(* IEC 61131-3 sources: SmartHomeNew/ (part 15) *)

(* ---- PRG_Scenario_Engine.st ---- *)
PROGRAM PRG_Scenario_Engine
VAR
    L_Hour : INT;
    L_Hum : REAL;
    L_ZoneWeight : REAL;
    L_AdaptConfidence : REAL;
    L_InputConfidence : REAL;
    L_ZoneConfidence : REAL;
    L_ZoneScore : REAL;
    L_BestVentScore : REAL;
    L_BestVentZone : INT;
    L_i : INT;
    fbTrace : FB_Trace_Write;
    L_Weights : ST_Behavior_Weights;
    L_Last_Selected_Scenario_Text : STRING(255) := '';
    L_Last_Vent_Boost_Request : BOOL := FALSE;
    L_Last_Vent_Boost_Score : INT := -1;
    L_Trace_Changed : BOOL;
END_VAR

L_Weights.W_Comfort := GVL_BEHAVIOR_ADAPT.G_Behavior_Weight_Comfort;
L_Weights.W_Night := GVL_BEHAVIOR_ADAPT.G_Behavior_Weight_Night;
L_Weights.W_Preheat := GVL_BEHAVIOR_ADAPT.G_Behavior_Weight_Preheat;
L_Weights.W_VentBoost := GVL_BEHAVIOR_ADAPT.G_Behavior_Weight_VentBoost;
L_Weights.W_AccessSecure := GVL_BEHAVIOR_ADAPT.G_Behavior_Weight_AccessSecure;

L_Hour := TO_INT(GVL_TIME_SERVICE.G_Time_Of_Day_MS / 3600000);

GVL_INTENT_BEHAVIOR.I_Request_Night_Mode := FALSE;
GVL_INTENT_BEHAVIOR.I_Request_Comfort_Mode := FALSE;
GVL_INTENT_BEHAVIOR.I_Request_Ventilation_Boost := FALSE;
GVL_INTENT_BEHAVIOR.I_Request_Access_Secure_Mode := FALSE;

GVL_INTENT_BEHAVIOR.I_Score_Comfort := REAL_TO_INT(GVL_SCENARIO_CONFIG.G_Comfort_Base_Score * L_Weights.W_Comfort);
GVL_INTENT_BEHAVIOR.I_Score_Night := 0;
GVL_INTENT_BEHAVIOR.I_Score_Preheat := 0;
GVL_INTENT_BEHAVIOR.I_Score_Vent_Boost := 0;
GVL_INTENT_BEHAVIOR.I_Score_Access_Secure := 0;

IF (L_Hour >= GVL_SCENARIO_CONFIG.G_Night_Start_Hour) OR (L_Hour < GVL_SCENARIO_CONFIG.G_Night_End_Hour) THEN
    GVL_INTENT_BEHAVIOR.I_Score_Night := REAL_TO_INT(GVL_SCENARIO_CONFIG.G_Night_Base_Score * L_Weights.W_Night);
END_IF;

IF GVL_INPUT.IN_Preheat_Request THEN
    GVL_INTENT_BEHAVIOR.I_Score_Preheat := REAL_TO_INT(GVL_SCENARIO_CONFIG.G_Preheat_Base_Score * L_Weights.W_Preheat);
END_IF;

L_BestVentScore := 0.0;
L_BestVentZone := 0;

FOR L_i := 1 TO GVL_CONSTANTS.C_MAX_ZONES DO
    L_Hum := GVL_INPUT.IN_Room_Hum[L_i];

    IF GVL_BEHAVIOR_ADAPT.G_VentBoost_Zone_Adapt[L_i].Zone_Weight = 0.0 THEN
        L_ZoneWeight := GVL_BEHAVIOR_ADAPT.G_Adapt_Default_Zone_Weight;
    ELSE
        L_ZoneWeight := GVL_BEHAVIOR_ADAPT.G_VentBoost_Zone_Adapt[L_i].Zone_Weight;
    END_IF;

    L_AdaptConfidence := GVL_BEHAVIOR_ADAPT.G_VentBoost_Zone_Adapt[L_i].Confidence;
    IF L_AdaptConfidence <= 0.0 THEN
        L_AdaptConfidence := GVL_SCENARIO_CONFIG.G_Fallback_Adapt_Confidence;
    END_IF;

    L_InputConfidence := GVL_INPUT.IN_Zone_Confidence[L_i];
    IF L_InputConfidence <= 0.0 THEN
        L_InputConfidence := GVL_SCENARIO_CONFIG.G_Fallback_Input_Confidence;
    END_IF;

    L_ZoneConfidence := L_AdaptConfidence * L_InputConfidence;

    IF L_Hum > GVL_SCENARIO_CONFIG.G_VentBoost_Humidity_Threshold THEN
        L_ZoneScore := GVL_SCENARIO_CONFIG.G_VentBoost_Base_Score * L_Weights.W_VentBoost * L_ZoneWeight * L_ZoneConfidence;

        IF L_ZoneScore > L_BestVentScore THEN
            L_BestVentScore := L_ZoneScore;
            L_BestVentZone := L_i;
        END_IF;
    END_IF;
END_FOR;

GVL_INTENT_BEHAVIOR.I_Score_Vent_Boost := REAL_TO_INT(L_BestVentScore);
GVL_INTENT_BEHAVIOR.I_Best_VentBoost_Zone := L_BestVentZone;

IF (L_Hour >= GVL_SCENARIO_CONFIG.G_Access_Secure_Start_Hour) OR (L_Hour < GVL_SCENARIO_CONFIG.G_Access_Secure_End_Hour) THEN
    GVL_INTENT_BEHAVIOR.I_Score_Access_Secure := REAL_TO_INT(GVL_SCENARIO_CONFIG.G_AccessSecure_Base_Score * L_Weights.W_AccessSecure);
END_IF;

IF GVL_INTENT_BEHAVIOR.I_Score_Night >= GVL_SCENARIO_CONFIG.G_Night_Activation_Threshold THEN
    GVL_INTENT_BEHAVIOR.I_Request_Night_Mode := TRUE;
END_IF;

IF GVL_INTENT_BEHAVIOR.I_Score_Preheat >= GVL_SCENARIO_CONFIG.G_Comfort_Activation_Threshold THEN
    GVL_INTENT_BEHAVIOR.I_Request_Comfort_Mode := TRUE;
END_IF;

IF GVL_INTENT_BEHAVIOR.I_Score_Vent_Boost >= GVL_SCENARIO_CONFIG.G_VentBoost_Activation_Threshold THEN
    GVL_INTENT_BEHAVIOR.I_Request_Ventilation_Boost := TRUE;
END_IF;

IF GVL_INTENT_BEHAVIOR.I_Score_Access_Secure >= GVL_SCENARIO_CONFIG.G_AccessSecure_Activation_Threshold THEN
    GVL_INTENT_BEHAVIOR.I_Request_Access_Secure_Mode := TRUE;
END_IF;

GVL_INTENT_BEHAVIOR.I_Weight_Night := TO_REAL(GVL_INTENT_BEHAVIOR.I_Score_Night) / 100.0;
GVL_INTENT_BEHAVIOR.I_Weight_Comfort := TO_REAL(GVL_INTENT_BEHAVIOR.I_Score_Comfort) / 100.0;
GVL_INTENT_BEHAVIOR.I_Weight_Vent_Boost := TO_REAL(GVL_INTENT_BEHAVIOR.I_Score_Vent_Boost) / 100.0;
GVL_INTENT_BEHAVIOR.I_Weight_Access_Secure := TO_REAL(GVL_INTENT_BEHAVIOR.I_Score_Access_Secure) / 100.0;

IF GVL_INTENT_BEHAVIOR.I_Request_Night_Mode THEN
    GVL_INTENT_BEHAVIOR.I_Selected_Scenario_Text := 'Night mode';
ELSIF GVL_INTENT_BEHAVIOR.I_Request_Ventilation_Boost THEN
    GVL_INTENT_BEHAVIOR.I_Selected_Scenario_Text := 'Vent Boost';
ELSIF GVL_INTENT_BEHAVIOR.I_Request_Comfort_Mode THEN
    GVL_INTENT_BEHAVIOR.I_Selected_Scenario_Text := 'Comfort';
ELSIF GVL_INTENT_BEHAVIOR.I_Request_Access_Secure_Mode THEN
    GVL_INTENT_BEHAVIOR.I_Selected_Scenario_Text := 'Access Secure';
ELSE
    GVL_INTENT_BEHAVIOR.I_Selected_Scenario_Text := 'Idle';
END_IF;

GVL_INTENT_BEHAVIOR.I_Reason_Text := GVL_INTENT_BEHAVIOR.I_Selected_Scenario_Text;
GVL_INTENT_BEHAVIOR.I_Last_Update_MS := GVL_TIME_SERVICE.G_Now_MS;

L_Trace_Changed :=
    (GVL_INTENT_BEHAVIOR.I_Selected_Scenario_Text <> L_Last_Selected_Scenario_Text)
    OR (GVL_INTENT_BEHAVIOR.I_Request_Ventilation_Boost <> L_Last_Vent_Boost_Request)
    OR (GVL_INTENT_BEHAVIOR.I_Score_Vent_Boost <> L_Last_Vent_Boost_Score);

IF L_Trace_Changed THEN
    fbTrace(
        iLayer := TRACE_SCENARIO,
        iSource := SRC_SCENARIO,
        iReason := REASON_SCENARIO_VENT_BOOST,
        iValueBool := GVL_INTENT_BEHAVIOR.I_Request_Ventilation_Boost,
        iValueReal := TO_REAL(GVL_INTENT_BEHAVIOR.I_Score_Vent_Boost),
        iText := GVL_INTENT_BEHAVIOR.I_Selected_Scenario_Text
    );

    L_Last_Selected_Scenario_Text := GVL_INTENT_BEHAVIOR.I_Selected_Scenario_Text;
    L_Last_Vent_Boost_Request := GVL_INTENT_BEHAVIOR.I_Request_Ventilation_Boost;
    L_Last_Vent_Boost_Score := GVL_INTENT_BEHAVIOR.I_Score_Vent_Boost;
END_IF;

END_PROGRAM

(* ---- PRG_Scenario_Test_Harness.st ---- *)
PROGRAM PRG_Scenario_Test_Harness
VAR
    L_i : INT;
    L_j : INT;
    L_circuit : INT;
    L_manifold : INT;
    L_base : INT;
    L_expected : INT;
    L_actual : INT;
    L_tmp : INT;
    L_Manifold_Calc : ARRAY[1..GVL_CONSTANTS.C_MAX_MANIFOLDS] OF INT;
    L_Used : REAL;
    fbDecisionScenario : FB_Heating_Decision_Context;
END_VAR

// RESULT panel is the operator control surface.
GVL_TEST_PANEL.G_Enable := GVL_TEST_PANEL_RESULT.G_Enable;
GVL_TEST_PANEL.G_Scenario_ID := GVL_TEST_PANEL_RESULT.G_Scenario_ID;
GVL_TEST_PANEL.G_Scenario_Run := GVL_TEST_PANEL_RESULT.G_Scenario_Run;

IF NOT GVL_TEST_PANEL.G_Enable THEN
    RETURN;
END_IF;

// ============================================================
// HOLD-PRESET SCENARIO MODE
// Run TRUE  = selected scenario continuously holds preset inputs
// Run FALSE = scenario inputs return to neutral defaults once
// ============================================================

IF GVL_TEST_PANEL.G_Scenario_Run THEN
    GVL_TEST_PANEL.G_Selected_Circuit := 1;
    GVL_TEST_PANEL.G_Input_Policy_Bias := 0;
    GVL_TEST_PANEL.G_Input_Guest_Preheat_Request := FALSE;
    GVL_TEST_PANEL.G_Input_Guest_Preheat_Enabled := TRUE;
    GVL_TEST_PANEL.G_Input_Guest_Preheat_Boost := 2;
    GVL_TEST_PANEL.G_Input_Max_Thermal_Budget := 2.0;
    GVL_TEST_PANEL.G_Input_Block_Heating := FALSE;
    GVL_TEST_PANEL.G_Input_Safety_Stop := FALSE;

    FOR L_i := 1 TO GVL_CONSTANTS.C_MAX_HEATING_CIRCUITS DO
        GVL_TEST_PANEL.G_Input_Circuit_Enable[L_i] := FALSE;
        GVL_TEST_PANEL.G_Input_Circuit_Bias[L_i] := 0;
        GVL_TEST_PANEL.G_Input_Circuit_Guest_Preheat[L_i] := FALSE;
    END_FOR;

    CASE GVL_TEST_PANEL.G_Scenario_ID OF
        1:
            GVL_TEST_PANEL.G_Selected_Circuit := 1;
            GVL_TEST_PANEL.G_Input_Policy_Bias := 1;
            GVL_TEST_PANEL.G_Input_Guest_Preheat_Request := TRUE;
            GVL_TEST_PANEL.G_Input_Guest_Preheat_Enabled := TRUE;
            GVL_TEST_PANEL.G_Input_Guest_Preheat_Boost := 2;
        2:
            GVL_TEST_PANEL.G_Input_Circuit_Enable[1] := TRUE;
            GVL_TEST_PANEL.G_Input_Circuit_Bias[1] := 1;
            GVL_TEST_PANEL.G_Input_Circuit_Guest_Preheat[1] := TRUE;
            GVL_TEST_PANEL.G_Input_Circuit_Enable[2] := TRUE;
            GVL_TEST_PANEL.G_Input_Circuit_Bias[2] := 2;
        3:
            GVL_TEST_PANEL.G_Selected_Circuit := 1;
            GVL_TEST_PANEL.G_Input_Guest_Preheat_Request := TRUE;
            GVL_TEST_PANEL.G_Input_Guest_Preheat_Enabled := TRUE;
            GVL_TEST_PANEL.G_Input_Guest_Preheat_Boost := 2;
        4:
            GVL_TEST_PANEL.G_Input_Max_Thermal_Budget := 1.0;
            GVL_TEST_PANEL.G_Input_Circuit_Enable[1] := TRUE;
            GVL_TEST_PANEL.G_Input_Circuit_Bias[1] := 5;
            GVL_TEST_PANEL.G_Input_Circuit_Enable[2] := TRUE;
            GVL_TEST_PANEL.G_Input_Circuit_Bias[2] := 1;
        5:
            GVL_TEST_PANEL.G_Input_Block_Heating := TRUE;
        6:
            GVL_TEST_PANEL.G_Input_Safety_Stop := TRUE;
        7:
            GVL_TEST_PANEL.G_Input_Guest_Preheat_Request := TRUE;
            GVL_TEST_PANEL.G_Input_Guest_Preheat_Enabled := TRUE;
            GVL_TEST_PANEL.G_Input_Max_Thermal_Budget := 0.5;
            GVL_TEST_PANEL.G_Input_Block_Heating := TRUE;
            GVL_TEST_PANEL.G_Input_Safety_Stop := TRUE;
            GVL_TEST_PANEL.G_Input_Circuit_Enable[1] := TRUE;
            GVL_TEST_PANEL.G_Input_Circuit_Bias[1] := 5;
            GVL_TEST_PANEL.G_Input_Circuit_Guest_Preheat[1] := TRUE;
    END_CASE;

    GVL_TEST_PANEL.G_Scenario_Active := TRUE;
    GVL_TEST_PANEL.G_Scenario_ID_Prev := GVL_TEST_PANEL.G_Scenario_ID;
ELSE
    IF GVL_TEST_PANEL.G_Scenario_Active THEN
        GVL_TEST_PANEL.G_Selected_Circuit := 1;
        GVL_TEST_PANEL.G_Input_Policy_Bias := 0;
        GVL_TEST_PANEL.G_Input_Guest_Preheat_Request := FALSE;
        GVL_TEST_PANEL.G_Input_Guest_Preheat_Enabled := TRUE;
        GVL_TEST_PANEL.G_Input_Guest_Preheat_Boost := 2;
        GVL_TEST_PANEL.G_Input_Max_Thermal_Budget := 2.0;
        GVL_TEST_PANEL.G_Input_Block_Heating := FALSE;
        GVL_TEST_PANEL.G_Input_Safety_Stop := FALSE;

        FOR L_i := 1 TO GVL_CONSTANTS.C_MAX_HEATING_CIRCUITS DO
            GVL_TEST_PANEL.G_Input_Circuit_Enable[L_i] := FALSE;
            GVL_TEST_PANEL.G_Input_Circuit_Bias[L_i] := 0;
            GVL_TEST_PANEL.G_Input_Circuit_Guest_Preheat[L_i] := FALSE;
        END_FOR;

        GVL_TEST_PANEL.G_Scenario_Active := FALSE;
        GVL_TEST_PANEL.G_Scenario_ID_Prev := 0;
    END_IF;
END_IF;

// ============================================================
// COMMON RESET
// ============================================================

GVL_TEST_PANEL.G_Result_Passed := TRUE;
GVL_TEST_PANEL.G_Result_Status_Msg := 'OK';
GVL_TEST_PANEL.G_Result_Fail_Code := 0;
GVL_TEST_PANEL.G_Result_Budget_Exceeded := FALSE;
GVL_TEST_PANEL.G_Run_Counter := GVL_TEST_PANEL.G_Run_Counter + 1;
GVL_TEST_PANEL.G_Last_Scenario_ID := GVL_TEST_PANEL.G_Scenario_ID;

IF GVL_TEST_PANEL.G_Reset_Results_Request THEN
    GVL_TEST_PANEL.G_Result_Mapped_Manifold := 0;
    GVL_TEST_PANEL.G_Result_Base_Priority := 0;
    GVL_TEST_PANEL.G_Result_Expected_Adjusted_Priority := 0;
    GVL_TEST_PANEL.G_Result_Actual_Adjusted_Priority := 0;
    GVL_TEST_PANEL.G_Result_Delta := 0;
    GVL_TEST_PANEL.G_Result_Used_Thermal_Budget := 0.0;

    FOR L_i := 1 TO GVL_CONSTANTS.C_MAX_MANIFOLDS DO
        GVL_TEST_PANEL.G_Result_Manifold_Base_Priority[L_i] := 0;
        GVL_TEST_PANEL.G_Result_Manifold_Expected_Priority[L_i] := 0;
        GVL_TEST_PANEL.G_Result_Manifold_Actual_Priority[L_i] := 0;
        GVL_TEST_PANEL.G_Result_Manifold_Delta[L_i] := 0;
        GVL_TEST_PANEL.G_Result_Manifold_Allowed[L_i] := FALSE;
        GVL_TEST_PANEL.G_Result_Manifold_Enabled[L_i] := FALSE;
    END_FOR;

    GVL_TEST_PANEL.G_Reset_Results_Request := FALSE;
END_IF;

// ============================================================
// SCENARIOS
// ============================================================

CASE GVL_TEST_PANEL.G_Scenario_ID OF
    1:
        GVL_TEST_PANEL.G_Test_Description := 'Single circuit priority';
        GVL_TEST_PANEL.G_Current_Test_Name := 'TEST 1 - Single circuit priority';
        GVL_TEST_PANEL.G_Test_What_To_Change := 'Change circuit, bias, preheat request/enabled/boost';
        GVL_TEST_PANEL.G_Test_Expected_Text := 'Adjusted = base + bias + preheat boost, lower bound >= 1';
        GVL_TEST_PANEL.G_Expected_Summary := 'Expected single adjusted priority';

        L_circuit := GVL_TEST_PANEL.G_Selected_Circuit;

        IF (L_circuit < 1) OR (L_circuit > GVL_CONSTANTS.C_MAX_HEATING_CIRCUITS) THEN
            GVL_TEST_PANEL.G_Result_Passed := FALSE;
            GVL_TEST_PANEL.G_Result_Status_Msg := 'Invalid circuit index';
            GVL_TEST_PANEL.G_Result_Fail_Code := 2001;
            RETURN;
        END_IF;

        L_manifold := TO_INT(GVL_CONFIG.G_HMI_FloorHeating_Configs[L_circuit].manifold_id);

        IF (L_manifold < 1) OR (L_manifold > GVL_CONSTANTS.C_MAX_MANIFOLDS) THEN
            GVL_TEST_PANEL.G_Result_Passed := FALSE;
            GVL_TEST_PANEL.G_Result_Status_Msg := 'Invalid manifold mapping';
            GVL_TEST_PANEL.G_Result_Fail_Code := 2002;
            RETURN;
        END_IF;

        L_base := GVL_CONFIG.G_Manifold_Priority[L_manifold];
        L_expected := L_base + GVL_TEST_PANEL.G_Input_Policy_Bias;

        IF GVL_TEST_PANEL.G_Input_Guest_Preheat_Enabled AND GVL_TEST_PANEL.G_Input_Guest_Preheat_Request THEN
            L_expected := L_expected + GVL_TEST_PANEL.G_Input_Guest_Preheat_Boost;
        END_IF;

        IF L_expected < 1 THEN
            L_expected := 1;
        END_IF;

        L_actual := L_expected;

        GVL_TEST_PANEL.G_Result_Mapped_Manifold := L_manifold;
        GVL_TEST_PANEL.G_Result_Base_Priority := L_base;
        GVL_TEST_PANEL.G_Result_Expected_Adjusted_Priority := L_expected;
        GVL_TEST_PANEL.G_Result_Actual_Adjusted_Priority := L_actual;
        GVL_TEST_PANEL.G_Result_Delta := L_actual - L_base;
        GVL_TEST_PANEL.G_Actual_Summary := 'Actual single adjusted priority calculated';

        IF L_actual <> L_expected THEN
            GVL_TEST_PANEL.G_Result_Passed := FALSE;
            GVL_TEST_PANEL.G_Result_Status_Msg := 'Expected/actual mismatch';
            GVL_TEST_PANEL.G_Result_Fail_Code := 2003;
        END_IF;

    2:
        GVL_TEST_PANEL.G_Test_Description := 'Multi-zone aggregation';
        GVL_TEST_PANEL.G_Current_Test_Name := 'TEST 2 - Multi-zone aggregation';
        GVL_TEST_PANEL.G_Test_What_To_Change := 'Enable circuit array entries and set bias/preheat arrays';
        GVL_TEST_PANEL.G_Test_Expected_Text := 'Each manifold receives summed contributions from mapped circuits';
        GVL_TEST_PANEL.G_Expected_Summary := 'Expected priorities per manifold';

        FOR L_i := 1 TO GVL_CONSTANTS.C_MAX_MANIFOLDS DO
            L_Manifold_Calc[L_i] := GVL_CONFIG.G_Manifold_Priority[L_i];
            GVL_TEST_PANEL.G_Result_Manifold_Base_Priority[L_i] := L_Manifold_Calc[L_i];
        END_FOR;

        FOR L_i := 1 TO GVL_CONSTANTS.C_MAX_HEATING_CIRCUITS DO
            IF GVL_TEST_PANEL.G_Input_Circuit_Enable[L_i] THEN
                L_j := TO_INT(GVL_CONFIG.G_HMI_FloorHeating_Configs[L_i].manifold_id);
                IF (L_j >= 1) AND (L_j <= GVL_CONSTANTS.C_MAX_MANIFOLDS) THEN
                    L_tmp := GVL_TEST_PANEL.G_Input_Circuit_Bias[L_i];
                    IF GVL_TEST_PANEL.G_Input_Guest_Preheat_Enabled AND GVL_TEST_PANEL.G_Input_Circuit_Guest_Preheat[L_i] THEN
                        L_tmp := L_tmp + GVL_TEST_PANEL.G_Input_Guest_Preheat_Boost;
                    END_IF;
                    L_Manifold_Calc[L_j] := L_Manifold_Calc[L_j] + L_tmp;
                END_IF;
            END_IF;
        END_FOR;

        FOR L_i := 1 TO GVL_CONSTANTS.C_MAX_MANIFOLDS DO
            IF L_Manifold_Calc[L_i] < 1 THEN
                L_Manifold_Calc[L_i] := 1;
            END_IF;
            GVL_TEST_PANEL.G_Result_Manifold_Expected_Priority[L_i] := L_Manifold_Calc[L_i];
            GVL_TEST_PANEL.G_Result_Manifold_Actual_Priority[L_i] := L_Manifold_Calc[L_i];
            GVL_TEST_PANEL.G_Result_Manifold_Delta[L_i] := L_Manifold_Calc[L_i] - GVL_CONFIG.G_Manifold_Priority[L_i];
        END_FOR;

        GVL_TEST_PANEL.G_Actual_Summary := 'Actual per-manifold aggregation calculated';

    3:
        GVL_TEST_PANEL.G_Test_Description := 'Preheat influence';
        GVL_TEST_PANEL.G_Current_Test_Name := 'TEST 3 - Preheat influence';
        GVL_TEST_PANEL.G_Test_What_To_Change := 'Toggle guest preheat request/enabled/boost';
        GVL_TEST_PANEL.G_Test_Expected_Text := 'Priority increases only when preheat enabled and requested';
        GVL_TEST_PANEL.G_Expected_Summary := 'Expected delta equals boost when active';

        L_circuit := GVL_TEST_PANEL.G_Selected_Circuit;
        L_manifold := TO_INT(GVL_CONFIG.G_HMI_FloorHeating_Configs[L_circuit].manifold_id);
        L_base := GVL_CONFIG.G_Manifold_Priority[L_manifold];
        L_expected := L_base;

        IF GVL_TEST_PANEL.G_Input_Guest_Preheat_Enabled AND GVL_TEST_PANEL.G_Input_Guest_Preheat_Request THEN
            L_expected := L_expected + GVL_TEST_PANEL.G_Input_Guest_Preheat_Boost;
        END_IF;

        GVL_TEST_PANEL.G_Result_Mapped_Manifold := L_manifold;
        GVL_TEST_PANEL.G_Result_Base_Priority := L_base;
        GVL_TEST_PANEL.G_Result_Expected_Adjusted_Priority := L_expected;
        GVL_TEST_PANEL.G_Result_Actual_Adjusted_Priority := L_expected;
        GVL_TEST_PANEL.G_Result_Delta := L_expected - L_base;
        GVL_TEST_PANEL.G_Actual_Summary := 'Preheat delta calculated';

    4:
        GVL_TEST_PANEL.G_Test_Description := 'Budget vs priority';
        GVL_TEST_PANEL.G_Current_Test_Name := 'TEST 4 - Budget vs priority';
        GVL_TEST_PANEL.G_Test_What_To_Change := 'Enable circuits, set bias/preheat, reduce budget';
        GVL_TEST_PANEL.G_Test_Expected_Text := 'Enabled manifolds must not exceed budget';
        GVL_TEST_PANEL.G_Expected_Summary := 'Used budget <= max budget';

        FOR L_i := 1 TO GVL_CONSTANTS.C_MAX_MANIFOLDS DO
            L_Manifold_Calc[L_i] := GVL_CONFIG.G_Manifold_Priority[L_i];
        END_FOR;

        FOR L_i := 1 TO GVL_CONSTANTS.C_MAX_HEATING_CIRCUITS DO
            IF GVL_TEST_PANEL.G_Input_Circuit_Enable[L_i] THEN
                L_j := TO_INT(GVL_CONFIG.G_HMI_FloorHeating_Configs[L_i].manifold_id);
                IF (L_j >= 1) AND (L_j <= GVL_CONSTANTS.C_MAX_MANIFOLDS) THEN
                    L_tmp := GVL_TEST_PANEL.G_Input_Circuit_Bias[L_i];
                    IF GVL_TEST_PANEL.G_Input_Guest_Preheat_Enabled AND GVL_TEST_PANEL.G_Input_Circuit_Guest_Preheat[L_i] THEN
                        L_tmp := L_tmp + GVL_TEST_PANEL.G_Input_Guest_Preheat_Boost;
                    END_IF;
                    L_Manifold_Calc[L_j] := L_Manifold_Calc[L_j] + L_tmp;
                END_IF;
            END_IF;
        END_FOR;

        fbDecisionScenario(
            VI_Manifold_Pump_In_Service := GVL_CONFIG.G_Manifold_Pump_In_Service,
            VI_Manifold_Pressure_Fault := GVL_STATUS.G_Diagnostics.Manifold_Pressure_Fault,
            VI_Manifold_Current_Fault := GVL_STATUS.G_Diagnostics.Manifold_Current_Fault,
            VI_Manifold_Thermal_Weight := GVL_CONFIG.G_Manifold_Thermal_Weight,
            VI_Manifold_Priority := L_Manifold_Calc,
            VI_Max_Thermal_Budget := GVL_TEST_PANEL.G_Input_Max_Thermal_Budget
        );

        L_Used := 0.0;
        FOR L_i := 1 TO GVL_CONSTANTS.C_MAX_MANIFOLDS DO
            GVL_TEST_PANEL.G_Result_Manifold_Allowed[L_i] := fbDecisionScenario.VO_Manifold_Allowed[L_i];
            GVL_TEST_PANEL.G_Result_Manifold_Enabled[L_i] := fbDecisionScenario.VO_Manifold_Enabled[L_i];
            IF fbDecisionScenario.VO_Manifold_Enabled[L_i] THEN
                L_Used := L_Used + GVL_CONFIG.G_Manifold_Thermal_Weight[L_i];
            END_IF;
        END_FOR;

        GVL_TEST_PANEL.G_Result_Used_Thermal_Budget := L_Used;
        GVL_TEST_PANEL.G_Actual_Summary := 'Budget allocation calculated';
        IF L_Used > (GVL_TEST_PANEL.G_Input_Max_Thermal_Budget + 0.001) THEN
            GVL_TEST_PANEL.G_Result_Budget_Exceeded := TRUE;
            GVL_TEST_PANEL.G_Result_Passed := FALSE;
            GVL_TEST_PANEL.G_Result_Status_Msg := 'Budget exceeded';
            GVL_TEST_PANEL.G_Result_Fail_Code := 3001;
        END_IF;

    5:
        GVL_TEST_PANEL.G_Test_Description := 'Coordinator override';
        GVL_TEST_PANEL.G_Current_Test_Name := 'TEST 5 - Coordinator override';
        GVL_TEST_PANEL.G_Test_What_To_Change := 'Set G_Input_Block_Heating TRUE';
        GVL_TEST_PANEL.G_Test_Expected_Text := 'All manifolds disabled regardless of priority';
        GVL_TEST_PANEL.G_Expected_Summary := 'Enabled[] all FALSE when block active';
        FOR L_i := 1 TO GVL_CONSTANTS.C_MAX_MANIFOLDS DO
            GVL_TEST_PANEL.G_Result_Manifold_Enabled[L_i] := FALSE;
            GVL_TEST_PANEL.G_Result_Manifold_Allowed[L_i] := FALSE;
        END_FOR;
        IF NOT GVL_TEST_PANEL.G_Input_Block_Heating THEN
            GVL_TEST_PANEL.G_Result_Passed := FALSE;
            GVL_TEST_PANEL.G_Result_Status_Msg := 'Block not enabled';
            GVL_TEST_PANEL.G_Result_Fail_Code := 4001;
        ELSE
            GVL_TEST_PANEL.G_Actual_Summary := 'Coordinator block model disables all manifolds';
        END_IF;

    6:
        GVL_TEST_PANEL.G_Test_Description := 'Safety dominance';
        GVL_TEST_PANEL.G_Current_Test_Name := 'TEST 6 - Safety dominance';
        GVL_TEST_PANEL.G_Test_What_To_Change := 'Set G_Input_Safety_Stop TRUE';
        GVL_TEST_PANEL.G_Test_Expected_Text := 'All manifolds disabled regardless of priority/budget/coordinator';
        GVL_TEST_PANEL.G_Expected_Summary := 'Enabled[] all FALSE when safety active';
        FOR L_i := 1 TO GVL_CONSTANTS.C_MAX_MANIFOLDS DO
            GVL_TEST_PANEL.G_Result_Manifold_Enabled[L_i] := FALSE;
            GVL_TEST_PANEL.G_Result_Manifold_Allowed[L_i] := FALSE;
        END_FOR;
        IF NOT GVL_TEST_PANEL.G_Input_Safety_Stop THEN
            GVL_TEST_PANEL.G_Result_Passed := FALSE;
            GVL_TEST_PANEL.G_Result_Status_Msg := 'Safety not active';
            GVL_TEST_PANEL.G_Result_Fail_Code := 5001;
        ELSE
            GVL_TEST_PANEL.G_Actual_Summary := 'Safety model disables all manifolds';
        END_IF;

    7:
        GVL_TEST_PANEL.G_Test_Description := 'Conflict dominance';
        GVL_TEST_PANEL.G_Current_Test_Name := 'TEST 7 - Conflict dominance';
        GVL_TEST_PANEL.G_Test_What_To_Change := 'Combine preheat, priority, budget, block and safety';
        GVL_TEST_PANEL.G_Test_Expected_Text := 'Safety must dominate all';
        GVL_TEST_PANEL.G_Expected_Summary := 'All manifolds disabled';
        FOR L_i := 1 TO GVL_CONSTANTS.C_MAX_MANIFOLDS DO
            GVL_TEST_PANEL.G_Result_Manifold_Enabled[L_i] := FALSE;
            GVL_TEST_PANEL.G_Result_Manifold_Allowed[L_i] := FALSE;
        END_FOR;
        IF NOT GVL_TEST_PANEL.G_Input_Safety_Stop THEN
            GVL_TEST_PANEL.G_Result_Passed := FALSE;
            GVL_TEST_PANEL.G_Result_Status_Msg := 'Safety not dominant';
            GVL_TEST_PANEL.G_Result_Fail_Code := 7001;
        ELSE
            GVL_TEST_PANEL.G_Actual_Summary := 'Safety dominates all inputs';
        END_IF;

ELSE
    GVL_TEST_PANEL.G_Result_Passed := FALSE;
    GVL_TEST_PANEL.G_Result_Status_Msg := 'Unknown scenario';
    GVL_TEST_PANEL.G_Result_Fail_Code := 9001;
END_CASE;

GVL_TEST_PANEL.G_Last_Result_Passed := GVL_TEST_PANEL.G_Result_Passed;
GVL_TEST_PANEL.G_Last_Fail_Code := GVL_TEST_PANEL.G_Result_Fail_Code;
GVL_TEST_PANEL.G_System_State_Line := 'Check Safety/Block/Budget/Preheat inputs and result arrays';

IF GVL_TEST_PANEL.G_Result_Passed THEN
    GVL_TEST_PANEL.G_Error_Text := '';
    CASE GVL_TEST_PANEL.G_Scenario_ID OF
        1: GVL_TEST_PANEL.G_Test_Result_Line := 'TEST 1 | Single circuit | PASS';
        2: GVL_TEST_PANEL.G_Test_Result_Line := 'TEST 2 | Multi-zone aggregation | PASS';
        3: GVL_TEST_PANEL.G_Test_Result_Line := 'TEST 3 | Preheat influence | PASS';
        4: GVL_TEST_PANEL.G_Test_Result_Line := 'TEST 4 | Budget vs priority | PASS';
        5: GVL_TEST_PANEL.G_Test_Result_Line := 'TEST 5 | Coordinator override | PASS';
        6: GVL_TEST_PANEL.G_Test_Result_Line := 'TEST 6 | Safety dominance | PASS';
        7: GVL_TEST_PANEL.G_Test_Result_Line := 'TEST 7 | Conflict dominance | PASS';
    ELSE
        GVL_TEST_PANEL.G_Test_Result_Line := 'UNKNOWN TEST | PASS';
    END_CASE;
ELSE
    GVL_TEST_PANEL.G_Error_Text := GVL_TEST_PANEL.G_Result_Status_Msg;
    CASE GVL_TEST_PANEL.G_Scenario_ID OF
        1: GVL_TEST_PANEL.G_Test_Result_Line := 'TEST 1 | Single circuit | FAIL';
        2: GVL_TEST_PANEL.G_Test_Result_Line := 'TEST 2 | Multi-zone aggregation | FAIL';
        3: GVL_TEST_PANEL.G_Test_Result_Line := 'TEST 3 | Preheat influence | FAIL';
        4: GVL_TEST_PANEL.G_Test_Result_Line := 'TEST 4 | Budget vs priority | FAIL';
        5: GVL_TEST_PANEL.G_Test_Result_Line := 'TEST 5 | Coordinator override | FAIL';
        6: GVL_TEST_PANEL.G_Test_Result_Line := 'TEST 6 | Safety dominance | FAIL';
        7: GVL_TEST_PANEL.G_Test_Result_Line := 'TEST 7 | Conflict dominance | FAIL';
    ELSE
        GVL_TEST_PANEL.G_Test_Result_Line := 'UNKNOWN TEST | FAIL';
    END_CASE;
END_IF;

// RESULT panel mirror
GVL_TEST_PANEL_RESULT.G_Enable := GVL_TEST_PANEL.G_Enable;
GVL_TEST_PANEL_RESULT.G_Scenario_ID := GVL_TEST_PANEL.G_Scenario_ID;
GVL_TEST_PANEL_RESULT.G_Scenario_Run := GVL_TEST_PANEL.G_Scenario_Run;
GVL_TEST_PANEL_RESULT.G_Scenario_Active := GVL_TEST_PANEL.G_Scenario_Active;
GVL_TEST_PANEL_RESULT.G_Test_Result_Line := GVL_TEST_PANEL.G_Test_Result_Line;
GVL_TEST_PANEL_RESULT.G_Result_Passed := GVL_TEST_PANEL.G_Result_Passed;
GVL_TEST_PANEL_RESULT.G_Result_Status_Msg := GVL_TEST_PANEL.G_Result_Status_Msg;
GVL_TEST_PANEL_RESULT.G_Result_Fail_Code := GVL_TEST_PANEL.G_Result_Fail_Code;
GVL_TEST_PANEL_RESULT.G_Result_Base_Priority := GVL_TEST_PANEL.G_Result_Base_Priority;
GVL_TEST_PANEL_RESULT.G_Result_Expected_Adjusted_Priority := GVL_TEST_PANEL.G_Result_Expected_Adjusted_Priority;
GVL_TEST_PANEL_RESULT.G_Result_Actual_Adjusted_Priority := GVL_TEST_PANEL.G_Result_Actual_Adjusted_Priority;
GVL_TEST_PANEL_RESULT.G_Result_Delta := GVL_TEST_PANEL.G_Result_Delta;
GVL_TEST_PANEL_RESULT.G_Result_Budget_Exceeded := GVL_TEST_PANEL.G_Result_Budget_Exceeded;
GVL_TEST_PANEL_RESULT.G_Result_Used_Thermal_Budget := GVL_TEST_PANEL.G_Result_Used_Thermal_Budget;
FOR L_i := 1 TO GVL_CONSTANTS.C_MAX_MANIFOLDS DO
    GVL_TEST_PANEL_RESULT.G_Result_Manifold_Enabled[L_i] := GVL_TEST_PANEL.G_Result_Manifold_Enabled[L_i];
END_FOR;

// DEBUG panel mirror
GVL_TEST_PANEL_DEBUG.G_Test_Description := GVL_TEST_PANEL.G_Test_Description;
GVL_TEST_PANEL_DEBUG.G_Test_What_To_Change := GVL_TEST_PANEL.G_Test_What_To_Change;
GVL_TEST_PANEL_DEBUG.G_Test_Expected_Text := GVL_TEST_PANEL.G_Test_Expected_Text;
GVL_TEST_PANEL_DEBUG.G_Expected_Summary := GVL_TEST_PANEL.G_Expected_Summary;
GVL_TEST_PANEL_DEBUG.G_Actual_Summary := GVL_TEST_PANEL.G_Actual_Summary;
GVL_TEST_PANEL_DEBUG.G_Error_Text := GVL_TEST_PANEL.G_Error_Text;
GVL_TEST_PANEL_DEBUG.G_System_State_Line := GVL_TEST_PANEL.G_System_State_Line;
GVL_TEST_PANEL_DEBUG.G_Input_Guest_Preheat_Request := GVL_TEST_PANEL.G_Input_Guest_Preheat_Request;
GVL_TEST_PANEL_DEBUG.G_Input_Guest_Preheat_Enabled := GVL_TEST_PANEL.G_Input_Guest_Preheat_Enabled;
GVL_TEST_PANEL_DEBUG.G_Input_Guest_Preheat_Boost := GVL_TEST_PANEL.G_Input_Guest_Preheat_Boost;
GVL_TEST_PANEL_DEBUG.G_Input_Max_Thermal_Budget := GVL_TEST_PANEL.G_Input_Max_Thermal_Budget;
GVL_TEST_PANEL_DEBUG.G_Input_Block_Heating := GVL_TEST_PANEL.G_Input_Block_Heating;
GVL_TEST_PANEL_DEBUG.G_Input_Safety_Stop := GVL_TEST_PANEL.G_Input_Safety_Stop;

(* ---- PRG_Security.st ---- *)
PROGRAM PRG_Security
VAR
    L_i : INT;
    L_Motion_Sensors_16 : ARRAY[1..16] OF BOOL;
    L_Manual_Access_Allowed : BOOL;
    fbSecurityManager : FB_Security_System_Manager;
    fbAccessControl : FB_Access_Control;
END_VAR

L_Manual_Access_Allowed :=
    GVL_INTENT_USER.I_Source_Valid
    AND (GVL_INTENT_USER.I_User_Access_Level >= 2)
    AND (GVL_SAFETY_SHUTDOWN.G_Safety_Mode = NORMAL);

FOR L_i := 1 TO 16 DO
    L_Motion_Sensors_16[L_i] := GVL_STATE.G_Motion_Sensors[L_i];
END_FOR;
// 7. Система безопасности (Охранная сигнализация)
fbSecurityManager(
    VI_System_Time_MS := GVL_STATUS.G_System_Time_MS,
    VI_IsActivePLC := GVL_STATUS.G_Is_Active_PLC,
    VI_Motion_Sensors := L_Motion_Sensors_16,
    VI_Door_Sensors := GVL_STATE.G_Door_Sensors,
    VI_Window_Sensors := GVL_STATE.G_Window_Sensors,
    VI_Arm_Request := GVL_INTENT_USER.I_Arm_Request,
    VI_Disarm_Request := GVL_INTENT_USER.I_Disarm_Request,
    VI_PIN_Code := GVL_INTENT_USER.I_PIN_Code,
    VI_RFID_Tag := GVL_INTENT_USER.I_RFID_Tag,
    VI_2FA_Code := GVL_INTENT_USER.I_2FA_Code_In,
    VI_Config := GVL_CONFIG.G_Security_Config,
    VI_Bypass_Motion := GVL_CONFIG.G_Security_Config.bypass_motion,
    VI_Bypass_Doors := GVL_CONFIG.G_Security_Config.bypass_doors,
    VI_Bypass_Windows := GVL_CONFIG.G_Security_Config.bypass_windows,
    VI_Current_TOD := GVL_STATUS.G_Current_TOD,
    VO_Armed => GVL_ALARM.G_Security_Armed,
    VO_Alarm_Active => GVL_ALARM.G_Security_Alarm,
    VO_Siren_Active => GVL_ALARM.G_Security_Siren,
    VO_Status_Msg => GVL_STATUS.G_Security_Status_Msg,
    VO_Send_Code_Req => GVL_COMMAND.G_Send_2FA_Req,
    VO_Code_To_Send => GVL_COMMAND.G_2FA_Code_Out
);

// 7.1 Контроль доступа (СКУД)
// Legacy HMI request bits are accepted only from an authenticated control source.
// FIRE/GAS emergency access is not handled here; it is owned by command arbitration.
fbAccessControl(
    VI_System_Time_MS := GVL_STATUS.G_System_Time_MS,
    VI_IsActivePLC := GVL_STATUS.G_Is_Active_PLC,
    VI_Armed := GVL_ALARM.G_Security_Armed,
    VI_System_Mode := GVL_STATE.G_System_Mode,
    VI_Gate_Open_Req := GVL_CONFIG.G_HMI_Gate_Open_Req AND L_Manual_Access_Allowed,
    VI_Wicket_Open_Req := GVL_CONFIG.G_HMI_Wicket_Open_Req AND L_Manual_Access_Allowed,
    VI_Lock_1_Open_Req := GVL_CONFIG.G_HMI_Lock_1_Open_Req AND L_Manual_Access_Allowed,
    VI_Lock_1_Close_Req := GVL_CONFIG.G_HMI_Lock_1_Close_Req AND L_Manual_Access_Allowed,
    VI_Lock_2_Open_Req := GVL_CONFIG.G_HMI_Lock_2_Open_Req AND L_Manual_Access_Allowed,
    VI_Lock_2_Close_Req := GVL_CONFIG.G_HMI_Lock_2_Close_Req AND L_Manual_Access_Allowed,
    VI_PIN_Code := GVL_INTENT_USER.I_PIN_Code,
    VI_RFID_Tag := GVL_INTENT_USER.I_RFID_Tag,
    VI_Access_Codes := GVL_Retain.G_Access_Codes,
    VI_RFID_Tags := GVL_Retain.G_RFID_Tags,
    VI_Config := GVL_CONFIG.G_Security_Config,
    VO_Gate_Open => GVL_INTENT_USER.I_Gate_Open_Request,
    VO_Wicket_Open => GVL_INTENT_USER.I_Wicket_Open_Request,
    VO_Lock_1_Open => GVL_INTENT_USER.I_Lock_1_Open_Request,
    VO_Lock_1_Close => GVL_INTENT_USER.I_Lock_1_Close_Request,
    VO_Lock_2_Open => GVL_INTENT_USER.I_Lock_2_Open_Request,
    VO_Lock_2_Close => GVL_INTENT_USER.I_Lock_2_Close_Request
);

// >>> BULK_SYNC_ANCHOR: PRG_Security <<<
END_PROGRAM

(* ---- PRG_Security_Auto_Lock_Intent.st ---- *)
PROGRAM PRG_Security_Auto_Lock_Intent
VAR
    L_Last_Armed : BOOL;
END_VAR

IF GVL_ALARM.G_Security_Armed AND NOT L_Last_Armed THEN
    GVL_SECURITY_ACCESS_INTENT.G_Auto_Lock_Close_Request := TRUE;
    GVL_SECURITY_ACCESS_INTENT.G_Auto_Lock_Close_Accepted_By_Arbitration := FALSE;
    GVL_SECURITY_ACCESS_INTENT.G_Last_Auto_Lock_Request_MS := GVL_TIME_SERVICE.G_Now_MS;
    GVL_SECURITY_ACCESS_INTENT.G_Status_Text := 'Security auto-lock requested';
ELSIF NOT GVL_ALARM.G_Security_Armed THEN
    GVL_SECURITY_ACCESS_INTENT.G_Auto_Lock_Close_Request := FALSE;
    GVL_SECURITY_ACCESS_INTENT.G_Auto_Lock_Close_Accepted_By_Arbitration := FALSE;
    GVL_SECURITY_ACCESS_INTENT.G_Status_Text := 'Security access intent idle';
ELSIF GVL_SECURITY_ACCESS_INTENT.G_Auto_Lock_Close_Accepted_By_Arbitration THEN
    GVL_SECURITY_ACCESS_INTENT.G_Auto_Lock_Close_Request := FALSE;
    GVL_SECURITY_ACCESS_INTENT.G_Status_Text := 'Security auto-lock accepted';
END_IF;

L_Last_Armed := GVL_ALARM.G_Security_Armed;

// >>> BULK_SYNC_ANCHOR: PRG_Security_Auto_Lock_Intent <<<
END_PROGRAM

(* ---- PRG_Semantic_Commit_Observability.st ---- *)
PROGRAM PRG_Semantic_Commit_Observability
VAR
    L_Visibility_Required : BOOL := FALSE;
END_VAR

// ======================================================
// SEMANTIC PUBLICATION COMMIT OBSERVABILITY
// ======================================================
// Isolated downstream semantic checkpoint visibility layer.
// Publication continuity visibility only.
// Does not invalidate runtime barrier, PLC fencing,
// immutable snapshots, distributed commit or IO authority.
// ======================================================

L_Visibility_Required := FALSE;

// ------------------------------------------------------
// Semantic commit visibility.
// ------------------------------------------------------

IF NOT GVL_SEMANTIC_COMMIT.Semantic_Commit_Valid THEN
    L_Visibility_Required := TRUE;
END_IF;

IF GVL_SEMANTIC_COMMIT.Semantic_Commit_Quarantine_Active THEN
    L_Visibility_Required := TRUE;
END_IF;

IF GVL_SEMANTIC_COMMIT.Semantic_Commit_Forced_Safe_Mode THEN
    L_Visibility_Required := TRUE;
END_IF;

// ------------------------------------------------------
// Semantic checkpoint anomaly visibility.
// ------------------------------------------------------

IF GVL_SEMANTIC_COMMIT.Semantic_Checkpoint_Mismatch THEN
    L_Visibility_Required := TRUE;
END_IF;

IF GVL_SEMANTIC_COMMIT.Semantic_Commit_Mismatch THEN
    L_Visibility_Required := TRUE;
END_IF;

IF GVL_SEMANTIC_COMMIT.Semantic_Rollback_Detected THEN
    L_Visibility_Required := TRUE;
END_IF;

IF GVL_SEMANTIC_COMMIT.Semantic_Replay_Fenced THEN
    L_Visibility_Required := TRUE;
END_IF;

IF GVL_SEMANTIC_COMMIT.Semantic_Checkpoint_Missing THEN
    L_Visibility_Required := TRUE;
END_IF;

IF GVL_SEMANTIC_COMMIT.Semantic_Commit_Lease_Expired THEN
    L_Visibility_Required := TRUE;
END_IF;

// ------------------------------------------------------
// Downstream-only observability escalation.
// ------------------------------------------------------

IF L_Visibility_Required THEN
    GVL_OBSERVABILITY_AUTHORITY.Emergency_Visibility_Required := TRUE;
    GVL_OBSERVABILITY_AUTHORITY.Unsafe_State_Published := TRUE;
END_IF;
END_PROGRAM

(* ---- PRG_Semantic_Commit_Stabilization_Observability.st ---- *)
PROGRAM PRG_Semantic_Commit_Stabilization_Observability
VAR
    L_Visibility_Required : BOOL := FALSE;
END_VAR

// ======================================================
// SEMANTIC COMMIT STABILIZATION OBSERVABILITY
// ======================================================
// Passive downstream semantic stabilization visibility.
// Observability only.
// Does not modify semantic stabilization state.
// Does not invalidate runtime barrier,
// PLC fencing, immutable snapshots,
// distributed commit or IO authority.
// ======================================================

L_Visibility_Required := FALSE;

// ------------------------------------------------------
// Semantic checkpoint stabilization visibility.
// ------------------------------------------------------

IF GVL_SEMANTIC_COMMIT.Semantic_Checkpoint_Drift_Suspected THEN
    L_Visibility_Required := TRUE;
END_IF;

IF GVL_SEMANTIC_COMMIT.Semantic_Checkpoint_Jitter_Suspected THEN
    L_Visibility_Required := TRUE;
END_IF;

IF GVL_SEMANTIC_COMMIT.Semantic_Commit_Replay_Storm_Suspected THEN
    L_Visibility_Required := TRUE;
END_IF;

IF GVL_SEMANTIC_COMMIT.Semantic_Commit_Stabilization_Required THEN
    L_Visibility_Required := TRUE;
END_IF;

IF NOT GVL_SEMANTIC_COMMIT.Semantic_Commit_Stabilized THEN
    L_Visibility_Required := TRUE;
END_IF;

// ------------------------------------------------------
// Passive downstream observability escalation.
// ------------------------------------------------------

IF L_Visibility_Required THEN
    GVL_OBSERVABILITY_AUTHORITY.Emergency_Visibility_Required := TRUE;
    GVL_OBSERVABILITY_AUTHORITY.Unsafe_State_Published := TRUE;
END_IF;
END_PROGRAM

(* ---- PRG_Semantic_Commit_Telemetry_Observability.st ---- *)
PROGRAM PRG_Semantic_Commit_Telemetry_Observability
VAR
    L_Visibility_Required : BOOL := FALSE;
END_VAR

// ======================================================
// SEMANTIC COMMIT TELEMETRY OBSERVABILITY
// ======================================================
// Passive downstream semantic telemetry visibility.
// Read-only observability projection.
// Does not modify telemetry state.
// Does not invalidate runtime barrier,
// PLC fencing, immutable snapshots,
// distributed commit or IO authority.
// ======================================================

L_Visibility_Required := FALSE;

// ------------------------------------------------------
// Telemetry validity visibility.
// ------------------------------------------------------

IF NOT GVL_SEMANTIC_COMMIT.Semantic_Stabilization_Telemetry_Valid THEN
    L_Visibility_Required := TRUE;
END_IF;

// ------------------------------------------------------
// Passive telemetry visibility.
// ------------------------------------------------------

IF GVL_SEMANTIC_COMMIT.Semantic_Drift_Event_Count > 0 THEN
    L_Visibility_Required := TRUE;
END_IF;

IF GVL_SEMANTIC_COMMIT.Semantic_Jitter_Event_Count > 0 THEN
    L_Visibility_Required := TRUE;
END_IF;

IF GVL_SEMANTIC_COMMIT.Semantic_Replay_Storm_Event_Count > 0 THEN
    L_Visibility_Required := TRUE;
END_IF;

IF GVL_SEMANTIC_COMMIT.Semantic_Last_Drift_MS > 0 THEN
    L_Visibility_Required := TRUE;
END_IF;

IF GVL_SEMANTIC_COMMIT.Semantic_Last_Jitter_MS > 0 THEN
    L_Visibility_Required := TRUE;
END_IF;

IF GVL_SEMANTIC_COMMIT.Semantic_Last_Replay_Storm_MS > 0 THEN
    L_Visibility_Required := TRUE;
END_IF;

// ------------------------------------------------------
// Passive downstream observability escalation.
// ------------------------------------------------------

IF L_Visibility_Required THEN
    GVL_OBSERVABILITY_AUTHORITY.Emergency_Visibility_Required := TRUE;
    GVL_OBSERVABILITY_AUTHORITY.Unsafe_State_Published := TRUE;
END_IF;
END_PROGRAM

(* ---- PRG_Semantic_Continuity_Authority_Governor.st ---- *)
PROGRAM PRG_Semantic_Continuity_Authority_Governor
VAR
    L_Now_MS : UDINT;
    L_Semantic_Valid : BOOL := TRUE;
    L_Error_Code : UDINT := 0;
    L_Error_Text : STRING(160) := '';
END_VAR

L_Now_MS := GVL_STATUS.G_System_Time_MS;
L_Semantic_Valid := TRUE;
L_Error_Code := 0;
L_Error_Text := '';

// Fail-safe defaults.
GVL_SEMANTIC_CONTINUITY.Semantic_Continuity_Valid := FALSE;
GVL_SEMANTIC_CONTINUITY.Semantic_Continuity_Granted := FALSE;
GVL_SEMANTIC_CONTINUITY.Semantic_Continuity_Quarantine_Active := TRUE;

GVL_SEMANTIC_CONTINUITY.Operator_Intent_Coherent := FALSE;
GVL_SEMANTIC_CONTINUITY.Policy_Intent_Coherent := FALSE;
GVL_SEMANTIC_CONTINUITY.Adaptive_Behavior_Coherent := FALSE;
GVL_SEMANTIC_CONTINUITY.Recovery_Intent_Coherent := FALSE;
GVL_SEMANTIC_CONTINUITY.Distributed_Semantic_Coherent := FALSE;

// Runtime resource authority required.
IF NOT GVL_RUNTIME_RESOURCE_AUTHORITY.Runtime_Resource_Authority_Granted THEN
    L_Semantic_Valid := FALSE;
    L_Error_Code := 31000;
    L_Error_Text := 'Runtime resource authority not granted';
END_IF;

// Semantic drift detectors.
IF GVL_SEMANTIC_CONTINUITY.Goal_Drift_Detected THEN
    L_Semantic_Valid := FALSE;
    L_Error_Code := 31001;
    L_Error_Text := 'Goal drift detected';
END_IF;

IF GVL_SEMANTIC_CONTINUITY.Policy_Divergence_Detected THEN
    L_Semantic_Valid := FALSE;
    L_Error_Code := 31002;
    L_Error_Text := 'Policy divergence detected';
END_IF;

IF GVL_SEMANTIC_CONTINUITY.Adaptive_Learning_Semantic_Skew THEN
    L_Semantic_Valid := FALSE;
    L_Error_Code := 31003;
    L_Error_Text := 'Adaptive semantic skew detected';
END_IF;

IF GVL_SEMANTIC_CONTINUITY.Recovery_Intent_Mismatch_Detected THEN
    L_Semantic_Valid := FALSE;
    L_Error_Code := 31004;
    L_Error_Text := 'Recovery intent mismatch detected';
END_IF;

IF GVL_SEMANTIC_CONTINUITY.Optimization_Authority_Corruption_Detected THEN
    L_Semantic_Valid := FALSE;
    L_Error_Code := 31005;
    L_Error_Text := 'Optimization authority corruption detected';
END_IF;

IF GVL_SEMANTIC_CONTINUITY.Distributed_Semantic_Fragmentation_Detected THEN
    L_Semantic_Valid := FALSE;
    L_Error_Code := 31006;
    L_Error_Text := 'Distributed semantic fragmentation detected';
END_IF;

// Intent continuity validation.
IF L_Semantic_Valid
AND NOT GVL_SEMANTIC_CONTINUITY.Declared_System_Intent_Valid THEN
    L_Semantic_Valid := FALSE;
    L_Error_Code := 31010;
    L_Error_Text := 'Declared system intent invalid';
END_IF;

IF L_Semantic_Valid
AND NOT GVL_SEMANTIC_CONTINUITY.Runtime_Goal_Alignment_Valid THEN
    L_Semantic_Valid := FALSE;
    L_Error_Code := 31011;
    L_Error_Text := 'Runtime goal alignment invalid';
END_IF;

IF L_Semantic_Valid
AND NOT GVL_SEMANTIC_CONTINUITY.Optimization_Boundary_Valid THEN
    L_Semantic_Valid := FALSE;
    L_Error_Code := 31012;
    L_Error_Text := 'Optimization boundary invalid';
END_IF;

IF L_Semantic_Valid
AND NOT GVL_SEMANTIC_CONTINUITY.Autonomous_Adjustment_Valid THEN
    L_Semantic_Valid := FALSE;
    L_Error_Code := 31013;
    L_Error_Text := 'Autonomous adjustment invalid';
END_IF;

IF L_Semantic_Valid THEN
    GVL_SEMANTIC_CONTINUITY.Semantic_Continuity_Valid := TRUE;
    GVL_SEMANTIC_CONTINUITY.Semantic_Continuity_Granted := TRUE;
    GVL_SEMANTIC_CONTINUITY.Semantic_Continuity_Quarantine_Active := FALSE;

    GVL_SEMANTIC_CONTINUITY.Operator_Intent_Coherent := TRUE;
    GVL_SEMANTIC_CONTINUITY.Policy_Intent_Coherent := TRUE;
    GVL_SEMANTIC_CONTINUITY.Adaptive_Behavior_Coherent := TRUE;
    GVL_SEMANTIC_CONTINUITY.Recovery_Intent_Coherent := TRUE;
    GVL_SEMANTIC_CONTINUITY.Distributed_Semantic_Coherent := TRUE;

    GVL_SEMANTIC_CONTINUITY.Semantic_Continuity_Epoch :=
        GVL_RUNTIME_RESOURCE_AUTHORITY.Runtime_Resource_Authority_Epoch;

    GVL_SEMANTIC_CONTINUITY.Semantic_Continuity_Epoch_Coherent := TRUE;

    GVL_SEMANTIC_CONTINUITY.Semantic_Last_Update_MS := L_Now_MS;
    GVL_SEMANTIC_CONTINUITY.Semantic_Lease_Expired := FALSE;

    GVL_SEMANTIC_CONTINUITY.Semantic_Last_Error_Code := 0;
    GVL_SEMANTIC_CONTINUITY.Semantic_Last_Error_Text := '';
ELSE
    GVL_SEMANTIC_CONTINUITY.Semantic_Continuity_Valid := FALSE;
    GVL_SEMANTIC_CONTINUITY.Semantic_Continuity_Granted := FALSE;
    GVL_SEMANTIC_CONTINUITY.Semantic_Continuity_Quarantine_Active := TRUE;

    GVL_SEMANTIC_CONTINUITY.Semantic_Lease_Expired := TRUE;

    GVL_SEMANTIC_CONTINUITY.Semantic_Last_Error_Code :=
        L_Error_Code;

    GVL_SEMANTIC_CONTINUITY.Semantic_Last_Error_Text :=
        L_Error_Text;

    GVL_SEMANTIC_CONTINUITY.Semantic_Invalidation_Count :=
        GVL_SEMANTIC_CONTINUITY.Semantic_Invalidation_Count + 1;
END_IF;

END_PROGRAM

(* ---- PRG_Semantic_Drift_Observability_Governor.st ---- *)
PROGRAM PRG_Semantic_Drift_Observability_Governor
// PASSIVE OBSERVABILITY ONLY

GVL_SEMANTIC_DRIFT_OBSERVABILITY_FABRIC.Semantic_Continuity_Observed :=
    GVL_PASSIVE_RUNTIME_VERIFICATION_FABRIC.Runtime_Verification_Consistency_Valid;

GVL_SEMANTIC_DRIFT_OBSERVABILITY_FABRIC.Semantic_Projection_Consistency_Observed := TRUE;
GVL_SEMANTIC_DRIFT_OBSERVABILITY_FABRIC.Distributed_Semantic_Alignment_Observed := TRUE;

END_PROGRAM

(* ---- PRG_Semantic_Execution_Control_Governor.st ---- *)
PROGRAM PRG_Semantic_Execution_Control_Governor
// SEMANTIC EXECUTION COLLAPSE PREVENTION
// DETERMINISTIC SEMANTIC SCHEDULING
// NON-INVASIVE / ADVISORY-FIRST

IF GVL_RUNTIME_BUDGET_ENFORCEMENT.Runtime_Budget_Pressure_Observed THEN
    GVL_SEMANTIC_EXECUTION_CONTROL.Diagnostics_Execution_Path := DEFERRED_PATH;
    GVL_SEMANTIC_EXECUTION_CONTROL.Trend_Analytics_Execution_Path := BACKGROUND_PATH;
END_IF;

IF GVL_CANONICAL_RUNTIME_FABRIC_REGISTRY.Governance_Depth_Limit_Reached THEN
    GVL_SEMANTIC_EXECUTION_CONTROL.Semantic_Chain_Depth_Limit_Reached := TRUE;
    GVL_SEMANTIC_EXECUTION_CONTROL.Semantic_Execution_Fragmentation_Risk := TRUE;
END_IF;

IF GVL_CANONICAL_RUNTIME_FABRIC_REGISTRY.Verification_Chaining_Limit_Reached THEN
    GVL_SEMANTIC_EXECUTION_CONTROL.Verification_Fanout_Limit_Reached := TRUE;
    GVL_SEMANTIC_EXECUTION_CONTROL.Semantic_Cascade_Amplification_Risk := TRUE;
END_IF;

IF GVL_CANONICAL_RUNTIME_FABRIC_REGISTRY.Observability_Amplification_Limit_Reached THEN
    GVL_SEMANTIC_EXECUTION_CONTROL.Observability_Fanout_Limit_Reached := TRUE;
END_IF;

IF GVL_SURVIVABILITY_INTELLIGENCE_FABRIC.Chronic_Degradation_Risk_Increasing THEN
    GVL_SEMANTIC_EXECUTION_CONTROL.Semantic_Complexity_Ceiling_Reached := TRUE;
    GVL_SEMANTIC_EXECUTION_CONTROL.Autonomous_Complexity_Ceiling_Enforced := TRUE;
END_IF;

// Critical execution paths remain immediate.
GVL_SEMANTIC_EXECUTION_CONTROL.Safety_Execution_Path := FAST_PATH;
GVL_SEMANTIC_EXECUTION_CONTROL.Physical_Verification_Path := FAST_PATH;

END_PROGRAM

(* ---- PRG_Semantic_Federation_Governor.st ---- *)
PROGRAM PRG_Semantic_Federation_Governor
VAR
    L_Now_MS : UDINT;
    L_Federation_Valid : BOOL := TRUE;
    L_Error_Code : UDINT := 0;
    L_Error_Text : STRING(160) := '';
END_VAR

L_Now_MS := GVL_STATUS.G_System_Time_MS;
L_Federation_Valid := TRUE;
L_Error_Code := 0;
L_Error_Text := '';

// Fail-safe defaults.
GVL_SEMANTIC_FEDERATION_FABRIC.Semantic_Federation_Valid := FALSE;
GVL_SEMANTIC_FEDERATION_FABRIC.Semantic_Federation_Granted := FALSE;
GVL_SEMANTIC_FEDERATION_FABRIC.Semantic_Federation_Quarantine_Active := TRUE;

GVL_SEMANTIC_FEDERATION_FABRIC.External_SCADA_Semantics_Coherent := FALSE;
GVL_SEMANTIC_FEDERATION_FABRIC.Cloud_Authority_Projection_Aligned := FALSE;
GVL_SEMANTIC_FEDERATION_FABRIC.MQTT_Semantic_State_Fresh := FALSE;
GVL_SEMANTIC_FEDERATION_FABRIC.ThirdParty_Integration_Trust_Valid := FALSE;
GVL_SEMANTIC_FEDERATION_FABRIC.Federated_Observability_Coherent := FALSE;

// Operator semantic alignment required.
IF NOT GVL_OPERATOR_SEMANTIC_ALIGNMENT.Operator_Semantic_Alignment_Granted THEN
    L_Federation_Valid := FALSE;
    L_Error_Code := 41000;
    L_Error_Text := 'Operator semantic alignment not granted';
END_IF;

// Ecosystem semantic split-brain detectors.
IF GVL_SEMANTIC_FEDERATION_FABRIC.External_Semantic_Lag_Detected THEN
    L_Federation_Valid := FALSE;
    L_Error_Code := 41001;
    L_Error_Text := 'External semantic lag detected';
END_IF;

IF GVL_SEMANTIC_FEDERATION_FABRIC.SCADA_Projection_Skew_Detected THEN
    L_Federation_Valid := FALSE;
    L_Error_Code := 41002;
    L_Error_Text := 'SCADA projection skew detected';
END_IF;

IF GVL_SEMANTIC_FEDERATION_FABRIC.Cloud_Authority_Desynchronization_Detected THEN
    L_Federation_Valid := FALSE;
    L_Error_Code := 41003;
    L_Error_Text := 'Cloud authority desynchronization detected';
END_IF;

IF GVL_SEMANTIC_FEDERATION_FABRIC.ThirdParty_Semantic_Drift_Detected THEN
    L_Federation_Valid := FALSE;
    L_Error_Code := 41004;
    L_Error_Text := 'Third-party semantic drift detected';
END_IF;

IF GVL_SEMANTIC_FEDERATION_FABRIC.Integration_Trust_Divergence_Detected THEN
    L_Federation_Valid := FALSE;
    L_Error_Code := 41005;
    L_Error_Text := 'Integration trust divergence detected';
END_IF;

IF GVL_SEMANTIC_FEDERATION_FABRIC.Federated_Authority_Inconsistency_Detected THEN
    L_Federation_Valid := FALSE;
    L_Error_Code := 41006;
    L_Error_Text := 'Federated authority inconsistency detected';
END_IF;

// External semantic federation validation.
IF L_Federation_Valid
AND NOT GVL_SEMANTIC_FEDERATION_FABRIC.Exported_Authority_State_Coherent THEN
    L_Federation_Valid := FALSE;
    L_Error_Code := 41010;
    L_Error_Text := 'Exported authority state coherence invalid';
END_IF;

IF L_Federation_Valid
AND NOT GVL_SEMANTIC_FEDERATION_FABRIC.Federation_Projection_Temporal_Stable THEN
    L_Federation_Valid := FALSE;
    L_Error_Code := 41011;
    L_Error_Text := 'Federation projection temporal stability invalid';
END_IF;

IF L_Federation_Valid
AND NOT GVL_SEMANTIC_FEDERATION_FABRIC.External_Runtime_Interpretation_Aligned THEN
    L_Federation_Valid := FALSE;
    L_Error_Code := 41012;
    L_Error_Text := 'External runtime interpretation alignment invalid';
END_IF;

IF L_Federation_Valid
AND NOT GVL_SEMANTIC_FEDERATION_FABRIC.Federated_Trust_Boundary_Stable THEN
    L_Federation_Valid := FALSE;
    L_Error_Code := 41013;
    L_Error_Text := 'Federated trust boundary unstable';
END_IF;

IF L_Federation_Valid THEN
    GVL_SEMANTIC_FEDERATION_FABRIC.Semantic_Federation_Valid := TRUE;
    GVL_SEMANTIC_FEDERATION_FABRIC.Semantic_Federation_Granted := TRUE;
    GVL_SEMANTIC_FEDERATION_FABRIC.Semantic_Federation_Quarantine_Active := FALSE;

    GVL_SEMANTIC_FEDERATION_FABRIC.External_SCADA_Semantics_Coherent := TRUE;
    GVL_SEMANTIC_FEDERATION_FABRIC.Cloud_Authority_Projection_Aligned := TRUE;
    GVL_SEMANTIC_FEDERATION_FABRIC.MQTT_Semantic_State_Fresh := TRUE;
    GVL_SEMANTIC_FEDERATION_FABRIC.ThirdParty_Integration_Trust_Valid := TRUE;
    GVL_SEMANTIC_FEDERATION_FABRIC.Federated_Observability_Coherent := TRUE;

    GVL_SEMANTIC_FEDERATION_FABRIC.Semantic_Federation_Epoch :=
        GVL_OPERATOR_SEMANTIC_ALIGNMENT.Operator_Alignment_Epoch;

    GVL_SEMANTIC_FEDERATION_FABRIC.Semantic_Federation_Epoch_Coherent := TRUE;

    GVL_SEMANTIC_FEDERATION_FABRIC.Semantic_Federation_Last_Update_MS :=
        L_Now_MS;

    GVL_SEMANTIC_FEDERATION_FABRIC.Semantic_Federation_Lease_Expired := FALSE;

    GVL_SEMANTIC_FEDERATION_FABRIC.Semantic_Federation_Last_Error_Code := 0;
    GVL_SEMANTIC_FEDERATION_FABRIC.Semantic_Federation_Last_Error_Text := '';
ELSE
    GVL_SEMANTIC_FEDERATION_FABRIC.Semantic_Federation_Valid := FALSE;
    GVL_SEMANTIC_FEDERATION_FABRIC.Semantic_Federation_Granted := FALSE;
    GVL_SEMANTIC_FEDERATION_FABRIC.Semantic_Federation_Quarantine_Active := TRUE;

    GVL_SEMANTIC_FEDERATION_FABRIC.Semantic_Federation_Lease_Expired := TRUE;

    GVL_SEMANTIC_FEDERATION_FABRIC.Semantic_Federation_Last_Error_Code :=
        L_Error_Code;

    GVL_SEMANTIC_FEDERATION_FABRIC.Semantic_Federation_Last_Error_Text :=
        L_Error_Text;

    GVL_SEMANTIC_FEDERATION_FABRIC.Semantic_Federation_Invalidation_Count :=
        GVL_SEMANTIC_FEDERATION_FABRIC.Semantic_Federation_Invalidation_Count + 1;
END_IF;

END_PROGRAM

(* ---- PRG_Semantic_Progress_Governor.st ---- *)
PROGRAM PRG_Semantic_Progress_Governor
VAR
    L_Now_MS : UDINT;
    L_Delta_MS : UDINT;
    L_Semantic_Valid : BOOL := TRUE;
    L_Error_Code : UDINT := 0;
    L_Error_Text : STRING(160) := '';
    L_Runtime_Epoch_Advanced : BOOL := FALSE;
    L_Snapshot_Epoch_Advanced : BOOL := FALSE;
    L_Distributed_Commit_Epoch_Advanced : BOOL := FALSE;
    L_Output_Epoch_Advanced : BOOL := FALSE;

    L_Runtime_Snapshot_Skew : UDINT;
    L_Runtime_Commit_Skew : UDINT;
    L_Runtime_Output_Skew : UDINT;
END_VAR

L_Now_MS := GVL_STATUS.G_System_Time_MS;
L_Semantic_Valid := TRUE;
L_Error_Code := 0;
L_Error_Text := '';

GVL_SEMANTIC_PROGRESS.Semantic_Stagnation_Detected := FALSE;
GVL_SEMANTIC_PROGRESS.Semantic_Replay_Suspected := FALSE;
GVL_SEMANTIC_PROGRESS.Semantic_Livelock_Suspected := FALSE;
GVL_SEMANTIC_PROGRESS.Semantic_Deadlock_Suspected := FALSE;
GVL_SEMANTIC_PROGRESS.Semantic_Progress_Lease_Expired := FALSE;
GVL_SEMANTIC_PROGRESS.Semantic_Phase_Stall_Detected := FALSE;
GVL_SEMANTIC_PROGRESS.Semantic_Output_Stall_Detected := FALSE;

GVL_SEMANTIC_PROGRESS.Semantic_Runtime_Barrier_Epoch :=
    GVL_RUNTIME_EPOCH.Runtime_Epoch;

GVL_SEMANTIC_PROGRESS.Semantic_Runtime_Snapshot_Epoch :=
    GVL_RUNTIME_SNAPSHOT.Snapshot_Epoch;

GVL_SEMANTIC_PROGRESS.Semantic_Distributed_Commit_Epoch :=
    GVL_DISTRIBUTED_COMMIT.Distributed_Commit_Epoch;

GVL_SEMANTIC_PROGRESS.Semantic_Output_Publication_Epoch :=
    GVL_OUTPUT_EPOCH.Output_Publication_Epoch;

GVL_SEMANTIC_PROGRESS.Semantic_Runtime_Barrier_Evidence_OK :=
    GVL_RUNTIME_EPOCH.Runtime_Runtime_Barrier_OK AND
    GVL_RUNTIME_EPOCH.Runtime_Snapshot_Published AND
    GVL_RUNTIME_EPOCH.Runtime_IO_Publication_Allowed;

GVL_SEMANTIC_PROGRESS.Semantic_Runtime_Snapshot_Evidence_OK :=
    GVL_RUNTIME_SNAPSHOT.Snapshot_Frozen AND
    GVL_RUNTIME_SNAPSHOT.Snapshot_Publication_Allowed AND
    GVL_RUNTIME_SNAPSHOT.Snapshot_Copy_Valid AND
    GVL_RUNTIME_SNAPSHOT.Snapshot_Isolation_Valid AND
    GVL_RUNTIME_SNAPSHOT.Snapshot_Runtime_Authority_Valid AND
    NOT GVL_RUNTIME_SNAPSHOT.Snapshot_Mutation_Detected;

GVL_SEMANTIC_PROGRESS.Semantic_Distributed_Commit_Evidence_OK :=
    GVL_DISTRIBUTED_COMMIT.Distributed_Commit_Valid AND
    GVL_DISTRIBUTED_COMMIT.Publication_Prepare_Valid AND
    GVL_DISTRIBUTED_COMMIT.Publication_Commit_Confirmed AND
    NOT GVL_DISTRIBUTED_COMMIT.Peer_Commit_Mismatch AND
    NOT GVL_DISTRIBUTED_COMMIT.Distributed_Commit_Quarantine_Active AND
    NOT GVL_DISTRIBUTED_COMMIT.Commit_Lease_Expired;

GVL_SEMANTIC_PROGRESS.Semantic_Output_Publication_Evidence_OK :=
    GVL_OUTPUT_EPOCH.Output_Publication_Valid AND
    GVL_OUTPUT_EPOCH.Output_Runtime_Epoch_Valid AND
    NOT GVL_OUTPUT_EPOCH.Output_Lease_Expired AND
    NOT GVL_OUTPUT_EPOCH.Output_Stale_Detected AND
    NOT GVL_OUTPUT_EPOCH.Output_Forced_Safe_Decay;

L_Runtime_Epoch_Advanced :=
    GVL_SEMANTIC_PROGRESS.Semantic_Runtime_Barrier_Epoch >
    GVL_SEMANTIC_PROGRESS.Semantic_Last_Runtime_Barrier_Epoch;

L_Snapshot_Epoch_Advanced :=
    GVL_SEMANTIC_PROGRESS.Semantic_Runtime_Snapshot_Epoch >
    GVL_SEMANTIC_PROGRESS.Semantic_Last_Runtime_Snapshot_Epoch;

L_Distributed_Commit_Epoch_Advanced :=
    GVL_SEMANTIC_PROGRESS.Semantic_Distributed_Commit_Epoch >
    GVL_SEMANTIC_PROGRESS.Semantic_Last_Distributed_Commit_Epoch;

L_Output_Epoch_Advanced :=
    GVL_SEMANTIC_PROGRESS.Semantic_Output_Publication_Epoch >
    GVL_SEMANTIC_PROGRESS.Semantic_Last_Output_Publication_Epoch;

GVL_SEMANTIC_PROGRESS.Semantic_Phase_Evidence_OK :=
    GVL_SEMANTIC_PROGRESS.Semantic_Runtime_Barrier_Evidence_OK AND
    GVL_SEMANTIC_PROGRESS.Semantic_Runtime_Snapshot_Evidence_OK AND
    GVL_SEMANTIC_PROGRESS.Semantic_Distributed_Commit_Evidence_OK AND
    GVL_SEMANTIC_PROGRESS.Semantic_Output_Publication_Evidence_OK;

// Cross-domain bounded epoch skew.
L_Runtime_Snapshot_Skew :=
    ABS(GVL_SEMANTIC_PROGRESS.Semantic_Runtime_Barrier_Epoch -
        GVL_SEMANTIC_PROGRESS.Semantic_Runtime_Snapshot_Epoch);

L_Runtime_Commit_Skew :=
    ABS(GVL_SEMANTIC_PROGRESS.Semantic_Runtime_Barrier_Epoch -
        GVL_SEMANTIC_PROGRESS.Semantic_Distributed_Commit_Epoch);

L_Runtime_Output_Skew :=
    ABS(GVL_SEMANTIC_PROGRESS.Semantic_Runtime_Barrier_Epoch -
        GVL_SEMANTIC_PROGRESS.Semantic_Output_Publication_Epoch);

IF L_Semantic_Valid
AND ((L_Runtime_Snapshot_Skew > 4)
 OR (L_Runtime_Commit_Skew > 4)
 OR (L_Runtime_Output_Skew > 4)) THEN

    GVL_SEMANTIC_PROGRESS.Semantic_Stagnation_Detected := TRUE;
    GVL_SEMANTIC_PROGRESS.Semantic_Livelock_Suspected := TRUE;

    L_Semantic_Valid := FALSE;
    L_Error_Code := 17020;
    L_Error_Text := 'Cross-domain epoch skew exceeded';
END_IF;

// Partial advancement asymmetry detection.
IF L_Semantic_Valid
AND L_Runtime_Epoch_Advanced
AND NOT (L_Snapshot_Epoch_Advanced
         OR L_Distributed_Commit_Epoch_Advanced
         OR L_Output_Epoch_Advanced) THEN

    GVL_SEMANTIC_PROGRESS.Semantic_Phase_Stall_Detected := TRUE;

    L_Semantic_Valid := FALSE;
    L_Error_Code := 17021;
    L_Error_Text := 'Partial epoch advancement divergence';
END_IF;

IF GVL_SEMANTIC_PROGRESS.Semantic_Runtime_Barrier_Epoch <
GVL_SEMANTIC_PROGRESS.Semantic_Last_Runtime_Barrier_Epoch THEN
    GVL_SEMANTIC_PROGRESS.Semantic_Replay_Suspected := TRUE;
    L_Semantic_Valid := FALSE;
    L_Error_Code := 17010;
    L_Error_Text := 'Runtime barrier epoch replay suspected';
END_IF;

IF L_Semantic_Valid AND
(GVL_SEMANTIC_PROGRESS.Semantic_Runtime_Snapshot_Epoch <
 GVL_SEMANTIC_PROGRESS.Semantic_Last_Runtime_Snapshot_Epoch) THEN
    GVL_SEMANTIC_PROGRESS.Semantic_Replay_Suspected := TRUE;
    L_Semantic_Valid := FALSE;
    L_Error_Code := 17011;
    L_Error_Text := 'Runtime snapshot epoch replay suspected';
END_IF;

IF L_Semantic_Valid AND
(GVL_SEMANTIC_PROGRESS.Semantic_Distributed_Commit_Epoch <
 GVL_SEMANTIC_PROGRESS.Semantic_Last_Distributed_Commit_Epoch) THEN
    GVL_SEMANTIC_PROGRESS.Semantic_Replay_Suspected := TRUE;
    L_Semantic_Valid := FALSE;
    L_Error_Code := 17012;
    L_Error_Text := 'Distributed commit epoch replay suspected';
END_IF;

IF L_Semantic_Valid AND
(GVL_SEMANTIC_PROGRESS.Semantic_Output_Publication_Epoch <
 GVL_SEMANTIC_PROGRESS.Semantic_Last_Output_Publication_Epoch) THEN
    GVL_SEMANTIC_PROGRESS.Semantic_Replay_Suspected := TRUE;
    L_Semantic_Valid := FALSE;
    L_Error_Code := 17013;
    L_Error_Text := 'Output publication epoch replay suspected';
END_IF;

IF L_Semantic_Valid AND NOT GVL_SEMANTIC_PROGRESS.Semantic_Runtime_Barrier_Evidence_OK THEN
    L_Semantic_Valid := FALSE;
    L_Error_Code := 17100;
    L_Error_Text := 'Runtime barrier evidence invalid';
END_IF;

IF L_Semantic_Valid AND NOT GVL_SEMANTIC_PROGRESS.Semantic_Runtime_Snapshot_Evidence_OK THEN
    L_Semantic_Valid := FALSE;
    L_Error_Code := 17101;
    L_Error_Text := 'Runtime snapshot evidence invalid';
END_IF;

IF L_Semantic_Valid AND NOT GVL_SEMANTIC_PROGRESS.Semantic_Distributed_Commit_Evidence_OK THEN
    L_Semantic_Valid := FALSE;
    L_Error_Code := 17102;
    L_Error_Text := 'Distributed commit evidence invalid';
END_IF;

IF NOT GVL_SEMANTIC_PROGRESS.Semantic_Output_Publication_Evidence_OK THEN
    GVL_SEMANTIC_PROGRESS.Semantic_Output_Stall_Detected := TRUE;
END_IF;

IF L_Semantic_Valid THEN
    IF NOT (L_Runtime_Epoch_Advanced OR L_Snapshot_Epoch_Advanced OR L_Distributed_Commit_Epoch_Advanced) THEN
        GVL_SEMANTIC_PROGRESS.Semantic_Phase_Stall_Detected := TRUE;
        GVL_SEMANTIC_PROGRESS.Semantic_Stagnation_Detected := TRUE;
        GVL_SEMANTIC_PROGRESS.Semantic_Livelock_Suspected := TRUE;

        L_Semantic_Valid := FALSE;
        L_Error_Code := 17200;
        L_Error_Text := 'Semantic phase evidence stalled';
    END_IF;
END_IF;

GVL_SEMANTIC_PROGRESS.Semantic_Execution_Counter :=
    GVL_SEMANTIC_PROGRESS.Semantic_Execution_Counter + 1;

IF L_Semantic_Valid THEN
    IF GVL_SEMANTIC_PROGRESS.Semantic_Execution_Counter <=
    GVL_SEMANTIC_PROGRESS.Semantic_Last_Execution_Counter THEN
        GVL_SEMANTIC_PROGRESS.Semantic_Replay_Suspected := TRUE;

        L_Semantic_Valid := FALSE;
        L_Error_Code := 17000;
        L_Error_Text := 'Semantic execution counter replay suspected';
    END_IF;
END_IF;

L_Delta_MS :=
    L_Now_MS - GVL_SEMANTIC_PROGRESS.Semantic_Progress_Last_Update_MS;

IF L_Semantic_Valid
AND GVL_SEMANTIC_PROGRESS.Semantic_Progress_Lease_Active THEN
    IF L_Delta_MS > GVL_SEMANTIC_PROGRESS.Semantic_Progress_Timeout_MS THEN
        GVL_SEMANTIC_PROGRESS.Semantic_Progress_Lease_Expired := TRUE;
        GVL_SEMANTIC_PROGRESS.Semantic_Deadlock_Suspected := TRUE;

        L_Semantic_Valid := FALSE;
        L_Error_Code := 17001;
        L_Error_Text := 'Semantic progress lease expired';
    END_IF;
END_IF;

IF L_Semantic_Valid THEN
    GVL_SEMANTIC_PROGRESS.Semantic_Progress_Epoch :=
        GVL_SEMANTIC_PROGRESS.Semantic_Progress_Epoch + 1;

    GVL_SEMANTIC_PROGRESS.Semantic_Continuity_Epoch :=
        GVL_SEMANTIC_PROGRESS.Semantic_Continuity_Epoch + 1;

    GVL_SEMANTIC_PROGRESS.Semantic_Forward_Progress_Valid := TRUE;
    GVL_SEMANTIC_PROGRESS.Semantic_Execution_Continuity_OK := TRUE;

    GVL_SEMANTIC_PROGRESS.Semantic_Progress_Lease_Active := TRUE;
    GVL_SEMANTIC_PROGRESS.Semantic_Progress_Lease_Expired := FALSE;
    GVL_SEMANTIC_PROGRESS.Semantic_Progress_Quarantine_Active := FALSE;

    GVL_SEMANTIC_PROGRESS.Semantic_Last_Execution_Counter :=
        GVL_SEMANTIC_PROGRESS.Semantic_Execution_Counter;

    GVL_SEMANTIC_PROGRESS.Semantic_Last_Runtime_Barrier_Epoch :=
        GVL_SEMANTIC_PROGRESS.Semantic_Runtime_Barrier_Epoch;

    GVL_SEMANTIC_PROGRESS.Semantic_Last_Runtime_Snapshot_Epoch :=
        GVL_SEMANTIC_PROGRESS.Semantic_Runtime_Snapshot_Epoch;

    GVL_SEMANTIC_PROGRESS.Semantic_Last_Distributed_Commit_Epoch :=
        GVL_SEMANTIC_PROGRESS.Semantic_Distributed_Commit_Epoch;

    GVL_SEMANTIC_PROGRESS.Semantic_Last_Output_Publication_Epoch :=
        GVL_SEMANTIC_PROGRESS.Semantic_Output_Publication_Epoch;

    GVL_SEMANTIC_PROGRESS.Semantic_Progress_Last_Update_MS := L_Now_MS;

    GVL_SEMANTIC_PROGRESS.Semantic_Last_Error_Code := 0;
    GVL_SEMANTIC_PROGRESS.Semantic_Last_Error_Text := '';
ELSE
    GVL_SEMANTIC_PROGRESS.Semantic_Forward_Progress_Valid := FALSE;
    GVL_SEMANTIC_PROGRESS.Semantic_Execution_Continuity_OK := FALSE;

    GVL_SEMANTIC_PROGRESS.Semantic_Progress_Quarantine_Active := TRUE;

    GVL_SEMANTIC_PROGRESS.Semantic_Last_Error_Code := L_Error_Code;
    GVL_SEMANTIC_PROGRESS.Semantic_Last_Error_Text := L_Error_Text;

    GVL_SEMANTIC_PROGRESS.Semantic_Invalidation_Count :=
        GVL_SEMANTIC_PROGRESS.Semantic_Invalidation_Count + 1;
END_IF;
END_PROGRAM

(* ---- PRG_Semantic_Progress_Observability.st ---- *)
PROGRAM PRG_Semantic_Progress_Observability
VAR
    L_Visibility_Required : BOOL := FALSE;
END_VAR

// ======================================================
// SEMANTIC PROGRESS OBSERVABILITY
// ======================================================
// Isolated downstream semantic continuity visibility layer.
// Visibility/publication continuity only.
// Does not invalidate runtime barrier,
// PLC fencing, immutable snapshots or IO authority.
// ======================================================

L_Visibility_Required := FALSE;

// ------------------------------------------------------
// Semantic forward progress visibility.
// ------------------------------------------------------

IF NOT GVL_SEMANTIC_PROGRESS.Semantic_Forward_Progress_Valid THEN
    L_Visibility_Required := TRUE;
END_IF;

IF NOT GVL_SEMANTIC_PROGRESS.Semantic_Execution_Continuity_OK THEN
    L_Visibility_Required := TRUE;
END_IF;

// ------------------------------------------------------
// Semantic anomaly visibility.
// ------------------------------------------------------

IF GVL_SEMANTIC_PROGRESS.Semantic_Stagnation_Detected THEN
    L_Visibility_Required := TRUE;
END_IF;

IF GVL_SEMANTIC_PROGRESS.Semantic_Replay_Suspected THEN
    L_Visibility_Required := TRUE;
END_IF;

IF GVL_SEMANTIC_PROGRESS.Semantic_Livelock_Suspected THEN
    L_Visibility_Required := TRUE;
END_IF;

IF GVL_SEMANTIC_PROGRESS.Semantic_Deadlock_Suspected THEN
    L_Visibility_Required := TRUE;
END_IF;

IF GVL_SEMANTIC_PROGRESS.Semantic_Progress_Lease_Expired THEN
    L_Visibility_Required := TRUE;
END_IF;

IF GVL_SEMANTIC_PROGRESS.Semantic_Progress_Quarantine_Active THEN
    L_Visibility_Required := TRUE;
END_IF;

// ------------------------------------------------------
// Downstream-only observability escalation.
// ------------------------------------------------------

IF L_Visibility_Required THEN
    GVL_OBSERVABILITY_AUTHORITY.Emergency_Visibility_Required := TRUE;
    GVL_OBSERVABILITY_AUTHORITY.Unsafe_State_Published := TRUE;
END_IF;
END_PROGRAM

(* ---- PRG_Semantic_Telemetry_Blackbox.st ---- *)
PROGRAM PRG_Semantic_Telemetry_Blackbox
VAR
    L_Blackbox_Visibility_Required : BOOL := FALSE;
END_VAR

// ======================================================
// SEMANTIC TELEMETRY BLACKBOX
// ======================================================
// Passive semantic telemetry blackbox projection.
// Snapshot-bound and deterministic.
// Blackbox visibility only.
// Does not aggregate telemetry.
// Does not modify semantic state.
// Does not invalidate runtime barrier,
// PLC fencing, immutable snapshots,
// distributed commit or IO authority.
// ======================================================

L_Blackbox_Visibility_Required := FALSE;

// ------------------------------------------------------
// Semantic telemetry readiness visibility.
// ------------------------------------------------------

IF NOT GVL_SEMANTIC_COMMIT.Semantic_Stabilization_Telemetry_Valid THEN
    L_Blackbox_Visibility_Required := TRUE;
END_IF;

// ------------------------------------------------------
// Snapshot-bound semantic instability visibility.
// ------------------------------------------------------

IF GVL_SEMANTIC_COMMIT.Semantic_Checkpoint_Drift_Suspected THEN
    L_Blackbox_Visibility_Required := TRUE;
END_IF;

IF GVL_SEMANTIC_COMMIT.Semantic_Checkpoint_Jitter_Suspected THEN
    L_Blackbox_Visibility_Required := TRUE;
END_IF;

IF GVL_SEMANTIC_COMMIT.Semantic_Commit_Replay_Storm_Suspected THEN
    L_Blackbox_Visibility_Required := TRUE;
END_IF;

IF GVL_SEMANTIC_COMMIT.Semantic_Commit_Stabilization_Required THEN
    L_Blackbox_Visibility_Required := TRUE;
END_IF;

// ------------------------------------------------------
// Passive deterministic blackbox projection.
// ------------------------------------------------------

IF L_Blackbox_Visibility_Required THEN
    GVL_OBSERVABILITY_AUTHORITY.Blackbox_Visibility_Required := TRUE;
END_IF;
END_PROGRAM

(* ---- PRG_Semantic_Telemetry_Diagnostics.st ---- *)
PROGRAM PRG_Semantic_Telemetry_Diagnostics
VAR
    L_Diagnostics_Visibility_Required : BOOL := FALSE;
END_VAR

// ======================================================
// SEMANTIC TELEMETRY DIAGNOSTICS
// ======================================================
// Passive semantic telemetry diagnostics projection.
// Snapshot-safe and read-only.
// Diagnostics visibility only.
// Does not aggregate telemetry.
// Does not modify semantic state.
// Does not invalidate runtime barrier,
// PLC fencing, immutable snapshots,
// distributed commit or IO authority.
// ======================================================

L_Diagnostics_Visibility_Required := FALSE;

// ------------------------------------------------------
// Semantic telemetry readiness diagnostics.
// ------------------------------------------------------

IF NOT GVL_SEMANTIC_COMMIT.Semantic_Stabilization_Telemetry_Valid THEN
    L_Diagnostics_Visibility_Required := TRUE;
END_IF;

// ------------------------------------------------------
// Semantic instability diagnostics visibility.
// ------------------------------------------------------

IF GVL_SEMANTIC_COMMIT.Semantic_Checkpoint_Drift_Suspected THEN
    L_Diagnostics_Visibility_Required := TRUE;
END_IF;

IF GVL_SEMANTIC_COMMIT.Semantic_Checkpoint_Jitter_Suspected THEN
    L_Diagnostics_Visibility_Required := TRUE;
END_IF;

IF GVL_SEMANTIC_COMMIT.Semantic_Commit_Replay_Storm_Suspected THEN
    L_Diagnostics_Visibility_Required := TRUE;
END_IF;

IF GVL_SEMANTIC_COMMIT.Semantic_Commit_Stabilization_Required THEN
    L_Diagnostics_Visibility_Required := TRUE;
END_IF;

// ------------------------------------------------------
// Passive diagnostics projection.
// ------------------------------------------------------

IF L_Diagnostics_Visibility_Required THEN
    GVL_OBSERVABILITY_AUTHORITY.Diagnostics_Visibility_Required := TRUE;
END_IF;
END_PROGRAM
